{attribute 'qualified_only'}
VAR_GLOBAL
	fAnalogData : REAL;
	fTestDelta : REAL;
	bTrendStatus : BOOL;
END_VAR

VAR_GLOBAL CONSTANT
	aiTrendArrayMax : INT;
END_VAR

(* stored: Version 1.1.0.1
   GVL GVL_Data: Id {a8a74dbe-f2ef-4675-ac7b-b7871c2dcb76} *)
